// TIA Portal project "Prakticne-4" (V16)

(* hardware
DEVICE "S7-1200 station_1"  S7-1200 Station
   slot 0: "Rack_0"  S7-1200 Rack  Rack  V1.0
   slot 1: "PLC_1"  CPU 1214C AC/DC/Rly  6ES7 214-1BG31-0XB0  V3.0
*)

// ===== PLC "PLC_1"  CPU 1214C AC/DC/Rly =====

VAR_GLOBAL   // PLC tag table "Default tag table"
   "Clock_Byte" AT %MB10 : Byte;
   "Clock_10Hz" AT %M10.0 : Bool;
   "Clock_5Hz" AT %M10.1 : Bool;
   "Clock_2.5Hz" AT %M10.2 : Bool;
   "Clock_2Hz" AT %M10.3 : Bool;
   "Clock_1.25Hz" AT %M10.4 : Bool;
   "Clock_1Hz" AT %M10.5 : Bool;
   "Clock_0.625Hz" AT %M10.6 : Bool;
   "Clock_0.5Hz" AT %M10.7 : Bool;
   "Tag_1" AT %M20.0 : Bool;
   "Tag_2" AT %M30.1 : Bool;
   "Tag_3" AT %M30.2 : Bool;
   "Tag_4" AT %M40.0 : Bool;
   "Tag_5" AT %M45.1 : Bool;
   "Tag_6" AT %M60.1 : Bool;
   "Tag_7" AT %M70.1 : Bool;
END_VAR

VAR_GLOBAL   // PLC tag table "Tag table_1"
   "Prekidac 1" AT %I0.0 : Bool;
   "Prekidac 2" AT %I0.1 : Bool;
   "Prekidac 3" AT %I0.2 : Bool;
   "Prekidac 4" AT %I0.3 : Bool;
   "Prekidac 5" AT %I0.4 : Bool;
   "Prekidac 6" AT %I0.5 : Bool;
   "Prekidac 7" AT %I0.6 : Bool;
   "Induktivni senzor" AT %I1.0 : Bool;
   "Pun krig napravljen" AT %I1.1 : Bool;
   "Dioda 2" AT %Q0.0 : Bool;
   "Dioda 3" AT %Q0.1 : Bool;
   "Dioda 4" AT %Q0.2 : Bool;
   "Dioda 5" AT %Q0.3 : Bool;
   "Motor suprotno od kazaljke" AT %Q0.4 : Bool;
   "Motor u smeru kazaljke" AT %Q0.5 : Bool;
END_VAR

DATA_BLOCK "DB_stanja"   // DB1
{ S7_Optimized_Access := 'TRUE' }
VERSION : 0.1
   VAR
      Pokrenut_u_levo : Bool;
      Pokrenut_u_desno : Bool;
   END_VAR
BEGIN
END_DATA_BLOCK

DATA_BLOCK "DB_senzori_stanja"   // DB3
{ S7_Optimized_Access := 'TRUE' }
VERSION : 0.1
   VAR
      Pun_krug_rising : Bool;
      prekidac_za_paljenje_rising : Bool;
   END_VAR
BEGIN
END_DATA_BLOCK

// folder: System blocks/Program resources

DATA_BLOCK "DB_brojac_pomeraja_levo"   // DB2
{ S7_Optimized_Access := 'TRUE' }
AUTHOR : Simatic
FAMILY : IEC
NAME : CNTR
VERSION : 1.0
// stored: InstanceOfName IEC_COUNTER
"IEC_COUNTER"
BEGIN
END_DATA_BLOCK

DATA_BLOCK "DB_tajmer_pauza"   // DB4
{ S7_Optimized_Access := 'TRUE' }
AUTHOR : Simatic
FAMILY : IEC
NAME : IEC_TMR
VERSION : 1.0
// stored: InstanceOfName IEC_TIMER
"IEC_TIMER"
BEGIN
END_DATA_BLOCK

DATA_BLOCK "DB_brojac_pomeraja_desno"   // DB5
{ S7_Optimized_Access := 'TRUE' }
AUTHOR : Simatic
FAMILY : IEC
NAME : CNTR
VERSION : 1.0
// stored: InstanceOfName IEC_COUNTER
"IEC_COUNTER"
BEGIN
END_DATA_BLOCK

// folder: (top level)

FUNCTION "FC_kretanje" : Void   // FC1, LAD
{ S7_Optimized_Access := 'TRUE' }
VERSION : 0.1
   VAR_TEMP   // added for the SCL form of the ladder/FBD networks
      _w1 : Bool;
      _w2 : Bool;
   END_VAR
BEGIN

REGION Network 1
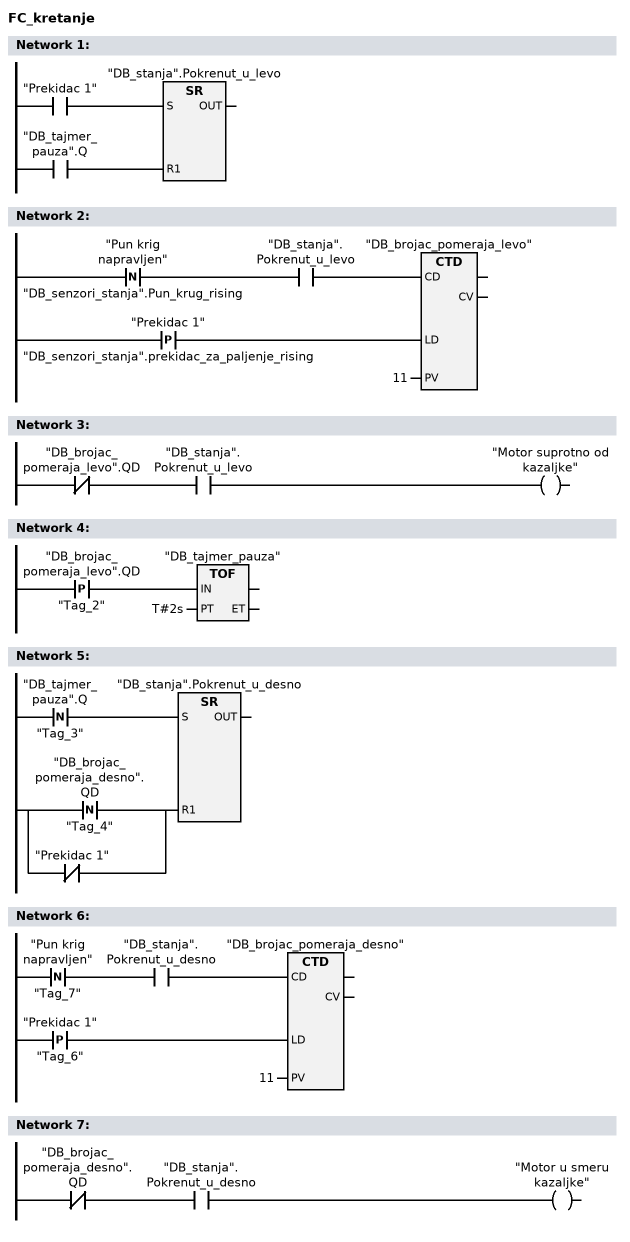
   RUNG wire#powerrail
      Contact( "Prekidac 1" )
      S_SR(operand := "DB_stanja".Pokrenut_u_levo, r1 := wire#w1)
   END_RUNG
   RUNG wire#powerrail
      Contact( "DB_tajmer_pauza".Q )
   END_RUNG wire#w1
   // the same network as SCL:
   IF "Prekidac 1" THEN
       "DB_stanja".Pokrenut_u_levo := TRUE;   // SR flip-flop
   END_IF;
   IF "DB_tajmer_pauza".Q THEN "DB_stanja".Pokrenut_u_levo := FALSE; END_IF;
END_REGION

REGION Network 2
   #_w1 := NOT "Pun krig napravljen" AND "DB_senzori_stanja".Pun_krug_rising;   // falling edge of "Pun krig napravljen"
   "DB_senzori_stanja".Pun_krug_rising := "Pun krig napravljen";
   #_w2 := "Prekidac 1" AND NOT "DB_senzori_stanja".prekidac_za_paljenje_rising;   // rising edge of "Prekidac 1"
   "DB_senzori_stanja".prekidac_za_paljenje_rising := "Prekidac 1";
   "DB_brojac_pomeraja_levo".CTD(CD := #_w1 AND "DB_stanja".Pokrenut_u_levo, LD := #_w2, PV := 11);
END_REGION

REGION Network 3
   RUNG wire#powerrail
      I_Contact( "DB_brojac_pomeraja_levo".QD )
      Contact( "DB_stanja".Pokrenut_u_levo )
      Coil( "Motor suprotno od kazaljke" )
   END_RUNG
   // the same network as SCL:
   "Motor suprotno od kazaljke" := NOT "DB_brojac_pomeraja_levo".QD AND "DB_stanja".Pokrenut_u_levo;
END_REGION

REGION Network 4
   #_w1 := "DB_brojac_pomeraja_levo".QD AND NOT "Tag_2";   // rising edge of "DB_brojac_pomeraja_levo".QD
   "Tag_2" := "DB_brojac_pomeraja_levo".QD;
   "DB_tajmer_pauza".TOF(IN := #_w1, PT := T#2s);
END_REGION

REGION Network 5
   RUNG wire#powerrail
      N_Contact(operand := "DB_tajmer_pauza".Q, bit := "Tag_3")
      S_SR(operand := "DB_stanja".Pokrenut_u_desno, r1 := wire#w1)
   END_RUNG
   RUNG wire#powerrail
      N_Contact(operand := "DB_brojac_pomeraja_desno".QD, bit := "Tag_4")
   END_RUNG wire#w1
   RUNG wire#powerrail
      I_Contact( "Prekidac 1" )
   END_RUNG wire#w1
   // the same network as SCL:
   #_w1 := NOT "DB_tajmer_pauza".Q AND "Tag_3";   // falling edge of "DB_tajmer_pauza".Q
   "Tag_3" := "DB_tajmer_pauza".Q;
   #_w2 := NOT "DB_brojac_pomeraja_desno".QD AND "Tag_4";   // falling edge of "DB_brojac_pomeraja_desno".QD
   "Tag_4" := "DB_brojac_pomeraja_desno".QD;
   IF #_w1 THEN
       "DB_stanja".Pokrenut_u_desno := TRUE;   // SR flip-flop
   END_IF;
   IF #_w2 OR NOT "Prekidac 1" THEN "DB_stanja".Pokrenut_u_desno := FALSE; END_IF;
END_REGION

REGION Network 6
   #_w1 := NOT "Pun krig napravljen" AND "Tag_7";   // falling edge of "Pun krig napravljen"
   "Tag_7" := "Pun krig napravljen";
   #_w2 := "Prekidac 1" AND NOT "Tag_6";   // rising edge of "Prekidac 1"
   "Tag_6" := "Prekidac 1";
   "DB_brojac_pomeraja_desno".CTD(CD := #_w1 AND "DB_stanja".Pokrenut_u_desno, LD := #_w2, PV := 11);
END_REGION

REGION Network 7
   RUNG wire#powerrail
      I_Contact( "DB_brojac_pomeraja_desno".QD )
      Contact( "DB_stanja".Pokrenut_u_desno )
      Coil( "Motor u smeru kazaljke" )
   END_RUNG
   // the same network as SCL:
   "Motor u smeru kazaljke" := NOT "DB_brojac_pomeraja_desno".QD AND "DB_stanja".Pokrenut_u_desno;
END_REGION
END_FUNCTION

ORGANIZATION_BLOCK "Main"   // OB1, LAD, ProgramCycle
TITLE = "Main Program Sweep (Cycle)"
{ S7_Optimized_Access := 'TRUE' }
VERSION : 0.1
BEGIN

REGION Network 1
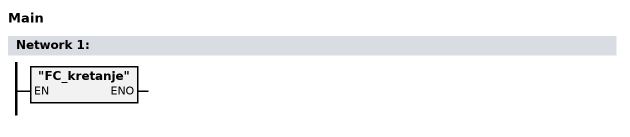
   RUNG wire#powerrail
      "FC_kretanje"()
   END_RUNG
   // the same network as SCL:
   "FC_kretanje"();
END_REGION
END_ORGANIZATION_BLOCK